Staubli VAL3: RecordAddon.pjx

--- RecordAddon.pjx ---
Parameters version=s7.9.1 stackSize=5000 millimeterUnit=true
Program file=start.pgx
Program file=stop.pgx
Data file=RecordAddon.dtx

--- RecordAddon.dtx ---
jointRx jJoint[3]
  [0] = {j1=-31.315744, j3=72.801072, j5=40.352904}
  [1] = {j1=-13.5, j3=72.801072, j5=40.352904}
  [2] = {j1=17.815744, j3=72.801072, j5=40.352904}
mdesc mNomSpeed
mdesc mSpeed = {accel=20, decel=20, tmax=100, blend=cartesian, leave=1, reach=1}

--- start.pgx ---
program start()
  local num l_ni
  local string l_sid
begin
  //清空储存器
  $recClean("c")
  //6轴，从1到6
  for l_ni=1 to 6
    l_sid="["+toString("",l_ni)+"]"
    //这里只是举例说明，不代表全部
    $recAdd("c","jntFbkPosErr"+l_sid)
    $recAdd("c","jntFbkFrc"+l_sid)
    $recAdd("c","jntFbkPos"+l_sid)
    $recAdd("c","jntCmdVel"+l_sid)
    $recAdd("c","jntFbkVel"+l_sid)
  endFor
  //
  movej(jJoint[0],flange,mSpeed)
  waitEndMove()
  //记录开始
  $recStart("c",30,250)
  delay(2)
  movej(jJoint[1],flange,mSpeed)
  movej(jJoint[2],flange,mSpeed)
  waitEndMove()
  delay(1)
  $recStop("c")
  //保存成文本文件。若保存成二进制文件："Disk://record"
  $recStore("ctt","Disk://record.txt")
end
